{attribute 'linkalways'} 
{attribute 'no_explicit_call' := 'This FB is a CLASS and must be accessed using methods or properties'}
{attribute 'enable_dynamic_creation'}
FUNCTION_BLOCK FINAL Node_REAL_TO_UDINT EXTENDS Node
VAR
	in : _REAL(0.0);
	out : _UDINT(0);
	success : _BOOL(FALSE);
END_VAR

METHOD PUBLIC  Clone : I_Node
VAR
	pNode : POINTER TO Node_REAL_TO_UDINT;
END_VAR
pNode := __NEW(Node_REAL_TO_UDINT);
Clone := pNode^;
END_METHOD

METHOD FB_init : BOOL
VAR_INPUT
	bInitRetains : BOOL; // if TRUE, the retain variables are initialized (warm start / cold start)
	bInCopyCode : BOOL;  // if TRUE, the instance afterwards gets moved into the copy code (online change)
END_VAR
AddParameter('in', in);
AddOutput('out', out);
AddOutput('success', success);

this^.Metadatum.AddBoolAsMetadata('deprecated', true);
END_METHOD

METHOD PROTECTED OnExecute
VAR
END_VAR
success.Value := TryConvert_REAL_TO_UDINT(in.Value, out.Value);
END_METHOD

END_FUNCTION_BLOCK

(* stored: Version 1.1.0.1, ProductVersion 3.1.4026.18
   POU Node_REAL_TO_UDINT: Id {dbe96478-017b-0646-3555-1a338d0c5e89}, SpecialFunc None
   Folder Constructor: Id {0aa86860-e342-05f6-0382-86a6b2c8a81d}
   Method Clone: Id {73bef8e9-46bf-0bef-2105-d1e1eedd4d87}
   Method FB_init: Id {8bab7f4e-c6b7-06be-0da7-6cb8e1e107bd}
   Method OnExecute: Id {4018701a-8554-0da0-3114-3c66f02059e2} *)
